// Mitsubishi GX Works2 project: 240514_MPSMxComponent   PLC: Q02U

PROGRAM MAIN
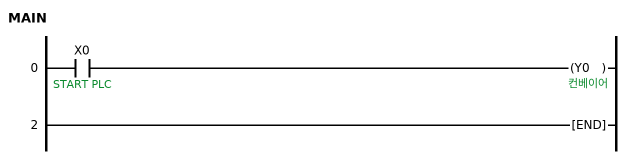
0     LD      X0  ; START PLC
      OUT     Y0  ; 컨베이어
2     END
END_PROGRAM

// device comments not shown above
X1  ; STOP PLC
Y1  ; RED LAMP
Y2  ; YELLOW LAMP
Y3  ; GREEN LAMP
Y4  ; 공급 감지 센서
Y5  ; 물체 감지 센서
Y6  ; 금속 감지 센서
Y10  ; 공급실린더 전진
Y11  ; 공급실린더 후진
Y12  ; 공급실린더 전진센서
Y13  ; 공급실린더 후진센서
Y20  ; 가공실린더 작동
Y22  ; 가공실린더 전진센서
Y23  ; 가공실린더 후진센서
Y30  ; 송출실린더 전진
Y31  ; 송출실린더 후진
Y32  ; 송출실린더 전진센서
Y33  ; 송출실린더 후진센서
Y40  ; 배출출실린더 전진
Y41  ; 배출실린더 후진
Y42  ; 배출실린더 전진센서
Y43  ; 배출실린더 후진센서
